// TwinCAT 3 PLC project PLC1
// ProgramVersion: 3.1.4023.0
// libraries:
//   Tc2_MC2, * (Beckhoff Automation GmbH)
//   Tc2_MC2_Drive, * (Beckhoff Automation GmbH)
//   Tc2_NcFifoAxes, * (Beckhoff Automation GmbH)
//   Tc2_Standard, * (Beckhoff Automation GmbH)
//   Tc2_System, * (Beckhoff Automation GmbH)
//   Tc2_Utilities, * (Beckhoff Automation GmbH)
//   Tc3_Module, * (Beckhoff Automation GmbH)
// project tree:
//   DUTs/ ST_streamOutputs.TcDUT
//   / PlcTask.TcTTO
//   POUs/ AxisBase.TcPOU, DigitalOut.TcPOU, FB_Fifo.TcPOU, FB_methods.TcPOU, FB_SetPositionBiasInNc_v1_10.TcPOU, FIFOaxis.TcPOU, FIFOIntegrate.TcPOU, IO.TcPOU, MAIN.TcPOU
// real-time tasks:
//   TASK PlcTask: cycle T#1ms, priority 20, ADS port 350
// motion (NC):
//   TASK NC-Task 1 SAF: cycle T#500us, priority 4, ADS port 501
//   TASK NC-Task 1 SVB: cycle T#1ms, priority 8, ADS port 511
//   AXIS motor_x1 (id 20)
//     OtherSettings: AllowMotionCmdToSlave=true, DataPersistence=true
//     encoder EncType=1
//     drive DrvType=5
//       Analog: TorqueSetpointScale=10, ScaleFactorActTorque=0.1
//       TimeComp: TaskDelayCycles=1
//     controller CtrType=1
//       CtrPara: PriorControlFactor=1
//         Observer: BandWidth=20
//   AXIS motor_x0 (id 1)
//     OtherSettings: AllowMotionCmdToSlave=true, DataPersistence=true
//     encoder EncType=1
//     drive DrvType=5
//       Analog: TorqueSetpointScale=10, ScaleFactorActTorque=0.1
//       TimeComp: TaskDelayCycles=1
//     controller CtrType=1
//       CtrPara: PriorControlFactor=1
//         Observer: BandWidth=20
//   AXIS motor_y0 (id 2)
//     OtherSettings: AllowMotionCmdToSlave=true, DataPersistence=true
//     encoder EncType=1
//     drive DrvType=5
//       Analog: TorqueSetpointScale=10, ScaleFactorActTorque=0.1
//       TimeComp: TaskDelayCycles=1
//     controller CtrType=1
//       CtrPara: PriorControlFactor=1
//         Observer: BandWidth=20
//   AXIS motor_y1 (id 3)
//     OtherSettings: AllowMotionCmdToSlave=true, DataPersistence=true
//     encoder EncType=1
//     drive DrvType=5
//       Analog: TorqueSetpointScale=10, ScaleFactorActTorque=0.1
//       TimeComp: TaskDelayCycles=1
//     controller CtrType=1
//       CtrPara: PriorControlFactor=1
//         Observer: BandWidth=20
//   AXIS motor_z1 (id 21)
//     OtherSettings: AllowMotionCmdToSlave=true, DataPersistence=true
//     encoder EncType=1
//     drive DrvType=5
//       Analog: TorqueSetpointScale=10, ScaleFactorActTorque=0.1
//       TimeComp: TaskDelayCycles=1
//     controller CtrType=1
//       CtrPara: PriorControlFactor=1
//         Observer: BandWidth=20
//   AXIS motor_z0 (id 4)
//     OtherSettings: AllowMotionCmdToSlave=true, DataPersistence=true
//     encoder EncType=1
//     drive DrvType=5
//       Analog: TorqueSetpointScale=10, ScaleFactorActTorque=0.1
//       TimeComp: TaskDelayCycles=1
//     controller CtrType=1
//       CtrPara: PriorControlFactor=1
//         Observer: BandWidth=20
//   AXIS motor_a0 (id 5)
//     OtherSettings: AllowMotionCmdToSlave=true, DataPersistence=true
//     encoder EncType=1
//     drive DrvType=5
//       Analog: TorqueSetpointScale=10, ScaleFactorActTorque=0.1
//       TimeComp: TaskDelayCycles=1
//     controller CtrType=1
//       CtrPara: PriorControlFactor=1
//         Observer: BandWidth=20
//   AXIS motor_b0 (id 6)
//     OtherSettings: AllowMotionCmdToSlave=true, DataPersistence=true
//     encoder EncType=1
//     drive DrvType=5
//       Analog: TorqueSetpointScale=10, ScaleFactorActTorque=0.1
//       TimeComp: TaskDelayCycles=1
//     controller CtrType=1
//       CtrPara: PriorControlFactor=1
//         Observer: BandWidth=20
//   AXIS motor_c0 (id 7)
//     OtherSettings: AllowMotionCmdToSlave=true, DataPersistence=true
//     encoder EncType=1
//     drive DrvType=5
//       Analog: TorqueSetpointScale=10, ScaleFactorActTorque=0.1
//       TimeComp: TaskDelayCycles=1
//     controller CtrType=1
//       CtrPara: PriorControlFactor=1
//         Observer: BandWidth=20
//   AXIS motor_d0 (id 8)
//     OtherSettings: AllowMotionCmdToSlave=true, DataPersistence=true
//     encoder EncType=1
//     drive DrvType=5
//       Analog: TorqueSetpointScale=10, ScaleFactorActTorque=0.1
//       TimeComp: TaskDelayCycles=1
//     controller CtrType=1
//       CtrPara: PriorControlFactor=1
//         Observer: BandWidth=20
//   AXIS motor_e0 (id 9)
//     OtherSettings: AllowMotionCmdToSlave=true, DataPersistence=true
//     encoder EncType=1
//     drive DrvType=5
//       Analog: TorqueSetpointScale=10, ScaleFactorActTorque=0.1
//       TimeComp: TaskDelayCycles=1
//     controller CtrType=1
//       CtrPara: PriorControlFactor=1
//         Observer: BandWidth=20
//   AXIS motor_x_master (id 10)
//     OtherSettings: AllowMotionCmdToSlave=true
//     encoder EncType=1
//     drive DrvType=5
//       Analog: TorqueSetpointScale=10, ScaleFactorActTorque=0.1
//       TimeComp: TaskDelayCycles=1
//     controller CtrType=1
//       CtrPara: PriorControlFactor=1
//         Observer: BandWidth=20
//   AXIS motor_y_master (id 11)
//     OtherSettings: AllowMotionCmdToSlave=true
//     encoder EncType=1
//     drive DrvType=5
//       Analog: TorqueSetpointScale=10, ScaleFactorActTorque=0.1
//       TimeComp: TaskDelayCycles=1
//     controller CtrType=1
//       CtrPara: PriorControlFactor=1
//         Observer: BandWidth=20
//   AXIS motor_z_master (id 12)
//     OtherSettings: AllowMotionCmdToSlave=true
//     encoder EncType=1
//     drive DrvType=5
//       Analog: TorqueSetpointScale=10, ScaleFactorActTorque=0.1
//       TimeComp: TaskDelayCycles=1
//     controller CtrType=1
//       CtrPara: PriorControlFactor=1
//         Observer: BandWidth=20
//   AXIS motor_a_master (id 13)
//     OtherSettings: AllowMotionCmdToSlave=true
//     encoder EncType=1
//     drive DrvType=5
//       Analog: TorqueSetpointScale=10, ScaleFactorActTorque=0.1
//       TimeComp: TaskDelayCycles=1
//     controller CtrType=1
//       CtrPara: PriorControlFactor=1
//         Observer: BandWidth=20
//   AXIS motor_b_master (id 14)
//     OtherSettings: AllowMotionCmdToSlave=true
//     encoder EncType=1
//     drive DrvType=5
//       Analog: TorqueSetpointScale=10, ScaleFactorActTorque=0.1
//       TimeComp: TaskDelayCycles=1
//     controller CtrType=1
//       CtrPara: PriorControlFactor=1
//         Observer: BandWidth=20
//   AXIS motor_c_master (id 15)
//     OtherSettings: AllowMotionCmdToSlave=true
//     encoder EncType=1
//     drive DrvType=5
//       Analog: TorqueSetpointScale=10, ScaleFactorActTorque=0.1
//       TimeComp: TaskDelayCycles=1
//     controller CtrType=1
//       CtrPara: PriorControlFactor=1
//         Observer: BandWidth=20
//   AXIS motor_d_master (id 16)
//     OtherSettings: AllowMotionCmdToSlave=true
//     encoder EncType=1
//     drive DrvType=5
//       Analog: TorqueSetpointScale=10, ScaleFactorActTorque=0.1
//       TimeComp: TaskDelayCycles=1
//     controller CtrType=1
//       CtrPara: PriorControlFactor=1
//         Observer: BandWidth=20
//   AXIS motor_e_master (id 17)
//     OtherSettings: AllowMotionCmdToSlave=true
//     encoder EncType=1
//     drive DrvType=5
//       Analog: TorqueSetpointScale=10, ScaleFactorActTorque=0.1
//       TimeComp: TaskDelayCycles=1
//     controller CtrType=1
//       CtrPara: PriorControlFactor=1
//         Observer: BandWidth=20
//   AXIS motor_z1_multimaster (id 22)
//     OtherSettings: AllowMotionCmdToSlave=true
//     encoder EncType=1
//     drive DrvType=5
//       Analog: TorqueSetpointScale=10, ScaleFactorActTorque=0.1
//       TimeComp: TaskDelayCycles=1
//     controller CtrType=1
//       CtrPara: PriorControlFactor=1
//         Observer: BandWidth=20
//   AXIS motor_z0_multimaster (id 18)
//     OtherSettings: AllowMotionCmdToSlave=true
//     encoder EncType=1
//     drive DrvType=5
//       Analog: TorqueSetpointScale=10, ScaleFactorActTorque=0.1
//       TimeComp: TaskDelayCycles=1
//     controller CtrType=1
//       CtrPara: PriorControlFactor=1
//         Observer: BandWidth=20
//   AXIS motor_z1_masterOffset (id 23)
//     OtherSettings: AllowMotionCmdToSlave=true
//     encoder EncType=1
//     drive DrvType=5
//       Analog: TorqueSetpointScale=10, ScaleFactorActTorque=0.1
//       TimeComp: TaskDelayCycles=1
//     controller CtrType=1
//       CtrPara: PriorControlFactor=1
//         Observer: BandWidth=20
//   AXIS motor_z0_masterOffset (id 19)
//     OtherSettings: AllowMotionCmdToSlave=true
//     encoder EncType=1
//     drive DrvType=5
//       Analog: TorqueSetpointScale=10, ScaleFactorActTorque=0.1
//       TimeComp: TaskDelayCycles=1
//     controller CtrType=1
//       CtrPara: PriorControlFactor=1
//         Observer: BandWidth=20
// variable links:
//   PLC1/PLC1 Instance <-> NC-Task 1 SAF/Axes/motor_a0
//     PlcTask Inputs/MAIN.motor_a0.axis.NcToPlc <-> Outputs/ToPlc
//     PlcTask Outputs/MAIN.motor_a0.axis.PlcToNc <-> Inputs/FromPlc
//   PLC1/PLC1 Instance <-> NC-Task 1 SAF/Axes/motor_a_master
//     PlcTask Inputs/MAIN.motor_a_master.axis.NcToPlc <-> Outputs/ToPlc
//     PlcTask Outputs/MAIN.motor_a_master.axis.PlcToNc <-> Inputs/FromPlc
//   PLC1/PLC1 Instance <-> NC-Task 1 SAF/Axes/motor_b0
//     PlcTask Inputs/MAIN.motor_b0.axis.NcToPlc <-> Outputs/ToPlc
//     PlcTask Outputs/MAIN.motor_b0.axis.PlcToNc <-> Inputs/FromPlc
//   PLC1/PLC1 Instance <-> NC-Task 1 SAF/Axes/motor_b_master
//     PlcTask Inputs/MAIN.motor_b_master.axis.NcToPlc <-> Outputs/ToPlc
//     PlcTask Outputs/MAIN.motor_b_master.axis.PlcToNc <-> Inputs/FromPlc
//   PLC1/PLC1 Instance <-> NC-Task 1 SAF/Axes/motor_c0
//     PlcTask Inputs/MAIN.motor_c0.axis.NcToPlc <-> Outputs/ToPlc
//     PlcTask Outputs/MAIN.motor_c0.axis.PlcToNc <-> Inputs/FromPlc
//   PLC1/PLC1 Instance <-> NC-Task 1 SAF/Axes/motor_c_master
//     PlcTask Inputs/MAIN.motor_c_master.axis.NcToPlc <-> Outputs/ToPlc
//     PlcTask Outputs/MAIN.motor_c_master.axis.PlcToNc <-> Inputs/FromPlc
//   PLC1/PLC1 Instance <-> NC-Task 1 SAF/Axes/motor_d0
//     PlcTask Inputs/MAIN.motor_d0.axis.NcToPlc <-> Outputs/ToPlc
//     PlcTask Outputs/MAIN.motor_d0.axis.PlcToNc <-> Inputs/FromPlc
//   PLC1/PLC1 Instance <-> NC-Task 1 SAF/Axes/motor_d_master
//     PlcTask Inputs/MAIN.motor_d_master.axis.NcToPlc <-> Outputs/ToPlc
//     PlcTask Outputs/MAIN.motor_d_master.axis.PlcToNc <-> Inputs/FromPlc
//   PLC1/PLC1 Instance <-> NC-Task 1 SAF/Axes/motor_e0
//     PlcTask Inputs/MAIN.motor_e0.axis.NcToPlc <-> Outputs/ToPlc
//     PlcTask Outputs/MAIN.motor_e0.axis.PlcToNc <-> Inputs/FromPlc
//   PLC1/PLC1 Instance <-> NC-Task 1 SAF/Axes/motor_e_master
//     PlcTask Inputs/MAIN.motor_e_master.axis.NcToPlc <-> Outputs/ToPlc
//     PlcTask Outputs/MAIN.motor_e_master.axis.PlcToNc <-> Inputs/FromPlc
//   PLC1/PLC1 Instance <-> NC-Task 1 SAF/Axes/motor_x0
//     PlcTask Inputs/MAIN.motor_x0.axis.NcToPlc <-> Outputs/ToPlc
//     PlcTask Outputs/MAIN.motor_x0.axis.PlcToNc <-> Inputs/FromPlc
//   PLC1/PLC1 Instance <-> NC-Task 1 SAF/Axes/motor_x1
//     PlcTask Inputs/MAIN.motor_x1.axis.NcToPlc <-> Outputs/ToPlc
//     PlcTask Outputs/MAIN.motor_x1.axis.PlcToNc <-> Inputs/FromPlc
//   PLC1/PLC1 Instance <-> NC-Task 1 SAF/Axes/motor_x_master
//     PlcTask Inputs/MAIN.motor_x_master.axis.NcToPlc <-> Outputs/ToPlc
//     PlcTask Outputs/MAIN.motor_x_master.axis.PlcToNc <-> Inputs/FromPlc
//   PLC1/PLC1 Instance <-> NC-Task 1 SAF/Axes/motor_y0
//     PlcTask Inputs/MAIN.motor_y0.axis.NcToPlc <-> Outputs/ToPlc
//     PlcTask Outputs/MAIN.motor_y0.axis.PlcToNc <-> Inputs/FromPlc
//   PLC1/PLC1 Instance <-> NC-Task 1 SAF/Axes/motor_y1
//     PlcTask Inputs/MAIN.motor_y1.axis.NcToPlc <-> Outputs/ToPlc
//     PlcTask Outputs/MAIN.motor_y1.axis.PlcToNc <-> Inputs/FromPlc
//   PLC1/PLC1 Instance <-> NC-Task 1 SAF/Axes/motor_y_master
//     PlcTask Inputs/MAIN.motor_y_master.axis.NcToPlc <-> Outputs/ToPlc
//     PlcTask Outputs/MAIN.motor_y_master.axis.PlcToNc <-> Inputs/FromPlc
//   PLC1/PLC1 Instance <-> NC-Task 1 SAF/Axes/motor_z0
//     PlcTask Inputs/MAIN.motor_z0.axis.NcToPlc <-> Outputs/ToPlc
//     PlcTask Outputs/MAIN.motor_z0.axis.PlcToNc <-> Inputs/FromPlc
//   PLC1/PLC1 Instance <-> NC-Task 1 SAF/Axes/motor_z0_masterOffset
//     PlcTask Inputs/MAIN.motor_z0_master_offset.axis.NcToPlc <-> Outputs/ToPlc
//     PlcTask Outputs/MAIN.motor_z0_master_offset.axis.PlcToNc <-> Inputs/FromPlc
//   PLC1/PLC1 Instance <-> NC-Task 1 SAF/Axes/motor_z0_multimaster
//     PlcTask Inputs/MAIN.motor_z0_multimaster.axis.NcToPlc <-> Outputs/ToPlc
//     PlcTask Outputs/MAIN.motor_z0_multimaster.axis.PlcToNc <-> Inputs/FromPlc
//   PLC1/PLC1 Instance <-> NC-Task 1 SAF/Axes/motor_z1
//     PlcTask Inputs/MAIN.motor_z1.axis.NcToPlc <-> Outputs/ToPlc
//     PlcTask Outputs/MAIN.motor_z1.axis.PlcToNc <-> Inputs/FromPlc
//   PLC1/PLC1 Instance <-> NC-Task 1 SAF/Axes/motor_z1_masterOffset
//     PlcTask Inputs/MAIN.motor_z1_master_offset.axis.NcToPlc <-> Outputs/ToPlc
//     PlcTask Outputs/MAIN.motor_z1_master_offset.axis.PlcToNc <-> Inputs/FromPlc
//   PLC1/PLC1 Instance <-> NC-Task 1 SAF/Axes/motor_z1_multimaster
//     PlcTask Inputs/MAIN.motor_z1_multimaster.axis.NcToPlc <-> Outputs/ToPlc
//     PlcTask Outputs/MAIN.motor_z1_multimaster.axis.PlcToNc <-> Inputs/FromPlc
//   PLC1/PLC1 Instance <-> NC-Task 1 SAF/Axes/motor_z_master
//     PlcTask Inputs/MAIN.motor_z_master.axis.NcToPlc <-> Outputs/ToPlc
//     PlcTask Outputs/MAIN.motor_z_master.axis.PlcToNc <-> Inputs/FromPlc

CONFIGURATION PLC1
    RESOURCE PLC ON TwinCAT3
        TASK PlcTask(INTERVAL := T#1ms, PRIORITY := 20);
        PROGRAM MAIN WITH PlcTask : MAIN;
    END_RESOURCE
END_CONFIGURATION

// ---- DUTs/ST_streamOutputs.TcDUT
TYPE ST_streamOutputs :
STRUCT
	cycleNo : UDINT;
	on : BOOL;

END_STRUCT
END_TYPE

// ---- POUs/MAIN.TcPOU
PROGRAM MAIN
VAR
	motor_x0 : AxisBase;
	motor_x1 : AxisBase;	
	motor_y0 : AxisBase;
	motor_y1 : AxisBase;
	motor_z0 : AxisBase;
	motor_z1 : AxisBase;	
	motor_a0 : AxisBase;
	motor_b0 : AxisBase;
	motor_c0 : AxisBase;
	motor_d0 : AxisBase;
	motor_e0 : AxisBase;
	
	motor_x_master : AxisBase;
	motor_y_master : AxisBase;
	motor_z_master : AxisBase;
	motor_a_master : AxisBase;
	motor_b_master : AxisBase;
	motor_c_master : AxisBase;
	motor_d_master : AxisBase;
	motor_e_master : AxisBase;
	
	motor_z0_master_offset : AxisBase;
	motor_z0_multimaster : AxisBase;
	motor_z1_master_offset : AxisBase;
	motor_z1_multimaster : AxisBase;
	emptyAxis1 : AXIS_REF;
	emptyAxis2 : AXIS_REF;

	gearOutAll: BOOL;
	n: INT;
	
	fbMultiMaster_z0 : MC_GearInMultiMaster;
	fbPower_multimaster : MC_Power;
	fbPower_z0_offset : MC_Power;
	bStartMultiMaster_z0: BOOL;
	fbGearOutMulti_z0 : MC_GearOut;
	
	fbMultiMaster_z1 : MC_GearInMultiMaster;
	fbPower_multimaster_z1 : MC_Power;
	fbPower_z1_offset : MC_Power;
	bStartMultiMaster_z1: BOOL;
	fbGearOutMulti_z1 : MC_GearOut;
	
	
	geartest : MC_GearIn;
	
	fbSystemTime : GETSYSTEMTIME;
	fileTime        : T_FILETIME;

	sTimeString: STRING(24);
	ppp: INT;
END_VAR


ppp := ppp + 1;


fbSystemTime(timeLoDW => fileTime.dwLowDateTime, timeHiDW => fileTime.dwHighDateTime );
sTimeString := SYSTEMTIME_TO_STRING(FILETIME_TO_SYSTEMTIME(fileTime));

FIFOaxis();

IO();


motor_x0(bPower:= , bMoveAbs:= , bMoveVel:= , bPowerStatus=> );
motor_x1(bPower:= , bMoveAbs:= , bMoveVel:= , bPowerStatus=> );
motor_y0(bPower:= , bMoveAbs:= , bMoveVel:= , bPowerStatus=> );
motor_y1(bPower:= , bMoveAbs:= , bMoveVel:= , bPowerStatus=> );
motor_z0(bPower:= , bMoveAbs:= , bMoveVel:= , bPowerStatus=> );
motor_z1(bPower:= , bMoveAbs:= , bMoveVel:= , bPowerStatus=> );
motor_a0(bPower:= , bMoveAbs:= , bMoveVel:= , bPowerStatus=> );
motor_b0(bPower:= , bMoveAbs:= , bMoveVel:= , bPowerStatus=> );
motor_c0(bPower:= , bMoveAbs:= , bMoveVel:= , bPowerStatus=> );
motor_d0(bPower:= , bMoveAbs:= , bMoveVel:= , bPowerStatus=> );
motor_e0(bPower:= , bMoveAbs:= , bMoveVel:= , bPowerStatus=> );

motor_x_master(bPower:= , bMoveAbs:= , bMoveVel:= , bPowerStatus=> );
motor_y_master(bPower:= , bMoveAbs:= , bMoveVel:= , bPowerStatus=> );
motor_z_master(bPower:= , bMoveAbs:= , bMoveVel:= , bPowerStatus=> );
motor_a_master(bPower:= , bMoveAbs:= , bMoveVel:= , bPowerStatus=> );
motor_b_master(bPower:= , bMoveAbs:= , bMoveVel:= , bPowerStatus=> );
motor_c_master(bPower:= , bMoveAbs:= , bMoveVel:= , bPowerStatus=> );
motor_d_master(bPower:= , bMoveAbs:= , bMoveVel:= , bPowerStatus=> );
motor_e_master(bPower:= , bMoveAbs:= , bMoveVel:= , bPowerStatus=> );

motor_z0_multimaster(bPower:= , bMoveAbs:= , bMoveVel:= , bPowerStatus=> );
motor_z0_master_offset(bPower:= , bMoveAbs:= , bMoveVel:= , bPowerStatus=> );
motor_z1_multimaster(bPower:= , bMoveAbs:= , bMoveVel:= , bPowerStatus=> );
motor_z1_master_offset(bPower:= , bMoveAbs:= , bMoveVel:= , bPowerStatus=> );




IF fbGearOutMulti_z0.Execute AND NOT fbGearOutMulti_z0.Busy THEN
	fbGearOutMulti_z0.Execute := FALSE;
END_IF
IF fbGearOutMulti_z1.Execute AND NOT fbGearOutMulti_z1.Busy THEN
	fbGearOutMulti_z1.Execute := FALSE;
END_IF

IF gearOutAll THEN
	bStartMultiMaster_z0 := FALSE;
	bStartMultiMaster_z1 := FALSE;	
	motor_x0.M_GearOut('motor_x0');
	motor_x1.M_GearOut('motor_x0');
	motor_y0.M_GearOut('motor_y0');
	motor_y1.M_GearOut('motor_y1');
	motor_z0.M_GearOut('motor_z0');
	motor_z1.M_GearOut('motor_z0');	
	motor_a0.M_GearOut('motor_a0');
	motor_b0.M_GearOut('motor_b0');
	motor_c0.M_GearOut('motor_c0');
	motor_d0.M_GearOut('motor_d0');
	motor_e0.M_GearOut('motor_e0');
	fbGearOutMulti_z0.Execute := TRUE;	
	fbGearOutMulti_z1.Execute := TRUE;	
	gearOutAll := FALSE;
END_IF




	
//multimaster, för z0-axel


fbMultiMaster_z0(
	Master1:= motor_z0_master_offset.axis, 
	Master2:= motor_z_master.axis, 
	Master3:= emptyAxis1, 
	Master4:= emptyAxis2, 
	Slave:= motor_z0_multimaster.axis, 
	Enable:= bStartMultiMaster_z0, 
	GearRatio1:= 1, 
	GearRatio2:= 1, 
	GearRatio3:= 0, 
	GearRatio4:= 0, 
	Acceleration:= , 
	Deceleration:= , 
	Jerk:= , 
	BufferMode:= , 
	Options:= , 
	InGear=> , 
	Busy=> , 
	Active=> , 
	CommandAborted=> , 
	Error=> , 
	ErrorID=> );

fbPower_multimaster(
	Axis:= motor_z0_multimaster.axis, 
	Enable:= TRUE, 
	Enable_Positive:= TRUE, 
	Enable_Negative:= TRUE, 
	Override:= , 
	BufferMode:= , 
	Options:= , 
	Status=> , 
	Busy=> , 
	Active=> , 
	Error=> , 
	ErrorID=> );

fbPower_z0_offset(
	Axis:= motor_z0_master_offset.axis, 
	Enable:= TRUE, 
	Enable_Positive:= TRUE, 
	Enable_Negative:= TRUE, 
	Override:= , 
	BufferMode:= , 
	Options:= , 
	Status=> , 
	Busy=> , 
	Active=> , 
	Error=> , 
	ErrorID=> );

fbGearOutMulti_z0(
	Slave:= motor_z0_multimaster.axis, 
	Execute:= , 
	Options:= , 
	Done=> , 
	Busy=> , 
	Error=> , 
	ErrorID=> );
	
	
//multimaster, för z1-axel


fbMultiMaster_z1(
	Master1:= motor_z1_master_offset.axis, 
	Master2:= motor_z_master.axis, 
	Master3:= emptyAxis1, 
	Master4:= emptyAxis2, 
	Slave:= motor_z1_multimaster.axis, 
	Enable:= bStartMultiMaster_z1, 
	GearRatio1:= 1, 
	GearRatio2:= 1, 
	GearRatio3:= 0, 
	GearRatio4:= 0, 
	Acceleration:= , 
	Deceleration:= , 
	Jerk:= , 
	BufferMode:= , 
	Options:= , 
	InGear=> , 
	Busy=> , 
	Active=> , 
	CommandAborted=> , 
	Error=> , 
	ErrorID=> );

fbPower_multimaster_z1(
	Axis:= motor_z1_multimaster.axis, 
	Enable:= TRUE, 
	Enable_Positive:= TRUE, 
	Enable_Negative:= TRUE, 
	Override:= , 
	BufferMode:= , 
	Options:= , 
	Status=> , 
	Busy=> , 
	Active=> , 
	Error=> , 
	ErrorID=> );

fbPower_z1_offset(
	Axis:= motor_z1_master_offset.axis, 
	Enable:= TRUE, 
	Enable_Positive:= TRUE, 
	Enable_Negative:= TRUE, 
	Override:= , 
	BufferMode:= , 
	Options:= , 
	Status=> , 
	Busy=> , 
	Active=> , 
	Error=> , 
	ErrorID=> );

fbGearOutMulti_z1(
	Slave:= motor_z1_multimaster.axis, 
	Execute:= , 
	Options:= , 
	Done=> , 
	Busy=> , 
	Error=> , 
	ErrorID=> );

METHOD M_GearOutAll : BOOL
VAR_INPUT
END_VAR
gearOutAll := TRUE;
END_METHOD

END_PROGRAM

// ---- POUs/AxisBase.TcPOU
FUNCTION_BLOCK AxisBase
VAR_INPUT
	bPower : BOOL;
	bMoveAbs : BOOL;
	bMoveVel : BOOL;

END_VAR
VAR_OUTPUT
	bPowerStatus : BOOL;
END_VAR
VAR
	isVirtual : BOOL;
	axis : AXIS_REF;
	fPosition : LREAL;		//from cnc
	fVelocity : LREAL;		//from cnc
	fAcc : LREAL;			//from cnc
	fDeacc : LREAL; 			//from cnc
	fbAxisPower : MC_Power;
	fbMoveAbsolute : MC_MoveAbsolute;
	fbHalt : MC_Halt;
	fbMoveVelocity : MC_MoveVelocity;
	axisState: INT;
	pp: INT;
	p: INT;
	fbGearIn : ARRAY[1..9] OF MC_GearIn;
	fbGearOut : MC_GearOut;
	a: INT;
	fbHome : MC_Home;
	fbHomeMemory: FB_CoEAX8000SetPositionOffset;  
	fbBias : FB_SetPositionBiasInNc_v1_10;  
	HomePos: LREAL;
	HomeSeq: INT;
	StartHome: BOOL;
	AxisHomed : BOOL;
	
	//torque
	MaxTorque : LREAL;
	MinTorque : LREAL;
	fbSoEread : FB_SoERead;
	
	axisIsGeared : BOOL;
	goBacktoFifo: BOOL;
	
	//reset
	fbReset : MC_Reset;
	b: INT;
	c: INT;
	fBias: LREAL;
	aa: INT;
	HomeSeqMemory: INT;
	StartHomeMemory: BOOL;
	bAxisDriveError: BOOL;
	bAxisError: BOOL;
END_VAR


axis.ReadStatus();
bAxisError:=axis.Status.Error;
bAxisDriveError:=axis.Status.DriveDeviceError;


CASE axisState OF

0:
	IF bMoveAbs THEN
		axisState := 100;
		b := b +1;
	END_IF
	IF bMoveVel THEN
		c := c +1;
		axisState := 200;
	END_IF

10:
	IF FIFOaxis.FifoActive THEN 
		goBacktoFifo := TRUE;
		MAIN.M_gearOutAll();
	END_IF	
	axisState := 20;

20:
	IF FIFOaxis.FifoActive THEN 
		FIFOaxis.M_deIntegrate();
	END_IF
	axisState := 30;
	

	
100:
	fbHalt.Execute := TRUE;
	IF (fbHalt.Busy AND NOT fbMoveAbsolute.Busy) OR fbHalt.Done THEN
		fbHalt.Execute := FALSE;
		axisState := 120;
	END_IF		

	
120:
	bMoveAbs := FALSE;	
	IF fVelocity <> 0 THEN
	fbmoveAbsolute.Execute := TRUE;
		axisState := 130;
	ELSE
		axisState := 0;
	END_IF
	
130:
	IF fbMoveAbsolute.Busy THEN
		fbMoveAbsolute.Execute := FALSE;
		axisState := 140;
	END_IF
	pp := pp +1;

140: 
	axisState := 0;	



200:
	fbHalt.Execute := TRUE;
	axisState := 210;

210:
	fbHalt.Execute := FALSE;
	axisState := 220;
	
220:
	bMoveVel := FALSE;
	IF fVelocity <> 0 THEN
		fbMoveVelocity.Execute := TRUE;	
		axisState := 230;
	ELSE
		axisState := 0;
	END_IF
	
230: 
	fbMoveVelocity.Execute := FALSE;
	axisState := 0;	


END_CASE





fbMoveAbsolute(
	Axis:= axis, 
	Execute:= , 
	Position:= fPosition, 
	Velocity:= fVelocity, 
	Acceleration:= fAcc, 
	Deceleration:= fDeacc, 
	Jerk:= 1000, 
	BufferMode:= ,//MC_BufferMode.MC_Aborting, 
	Options:= , 
	Done=> , 
	Busy=> , 
	Active=> , 
	CommandAborted=> , 
	Error=> , 
	ErrorID=> );
	
	
fbMoveVelocity(
	Axis:= axis, 
	Execute:= , 
	Velocity:= fVelocity, 
	Acceleration:= fAcc, 
	Deceleration:= fDeacc, 
	Jerk:= 5000, 
	Direction:= , 
	BufferMode:= , 
	Options:= , 
	InVelocity=> , 
	Busy=> , 
	Active=> , 
	CommandAborted=> , 
	Error=> , 
	ErrorID=> );

	
fbHalt(
	Axis:= axis, 
	Execute:= , 
	Deceleration:= 1000, 
	Jerk:= 5000, 
	BufferMode:= , 
	Options:= , 
	Done=> , 
	Busy=> , 
	Active=> , 
	CommandAborted=> , 
	Error=> , 
	ErrorID=> );

	
fbAxisPower(
	Axis:= axis, 
	Enable:= bPower, 
	Enable_Positive:= TRUE, 
	Enable_Negative:= TRUE, 
	Override:= 100, 
	BufferMode:= ,
	Options:= , 
	Status=> bPowerStatus, 
	Busy=> , 
	Active=> , 
	Error=> , 
	ErrorID=> );
	

	//GEAR

FOR a:=1 TO 9 DO
	IF fbGearIn[a].Execute AND fbGearIn[a].Busy THEN 
		fbGearIn[a].Execute := FALSE; 
	END_IF
END_FOR


IF fbGearOut.Execute AND fbGearOut.Busy THEN
	fbhalt.Execute := FALSE;
	fbGearOut.Execute := FALSE;
END_IF



	
fbGearOut(
	Slave:= axis, 
	Execute:= , 
	Options:= , 
	Done=> , 
	Busy=> , 
	Error=> , 
	ErrorID=> );

fbGearIn[1](Master:= main.motor_x_master.axis, Slave:= axis, RatioDenominator := 1, RatioNumerator := 1);
fbGearIn[2](Master:= main.motor_y_master.axis, Slave:= axis, RatioDenominator := 1, RatioNumerator := 1);
fbGearIn[3](Master:= main.motor_z0_multimaster.axis, Slave:= axis, RatioDenominator := 1, RatioNumerator := 1);
fbGearIn[4](Master:= main.motor_a_master.axis, Slave:= axis, RatioDenominator := 1, RatioNumerator := 1);
fbGearIn[5](Master:= main.motor_b_master.axis, Slave:= axis, RatioDenominator := 1, RatioNumerator := 1);
fbGearIn[6](Master:= main.motor_c_master.axis, Slave:= axis, RatioDenominator := 1, RatioNumerator := 1);
fbGearIn[7](Master:= main.motor_d_master.axis, Slave:= axis, RatioDenominator := 1, RatioNumerator := 1);
fbGearIn[8](Master:= main.motor_e_master.axis, Slave:= axis, RatioDenominator := 1, RatioNumerator := 1);
fbGearIn[9](Master:= main.motor_z1_multimaster.axis, Slave:= axis, RatioDenominator := 1, RatioNumerator := 1);	
	
//HOMING

CASE HomeSeq OF
	
	0: 
		IF 	StartHome THEN
			HomeSeq := 10;
		END_IF

		
	10:
		StartHome := FALSE;
		fbHome.Position := HomePos;
		HomeSeq := 20;
				aa := aa +1;
	20:
		fbHome.Execute := TRUE;
		//fbBias.bExecute :=TRUE;
		HomeSeq := 30;
		
	30:
		IF fbHome.Execute AND NOT fbHome.Busy THEN
			fbHome.Execute := FALSE;
			//fbBias.bExecute :=FALSE;
			HomeSeq :=0;
			AxisHomed := TRUE;
		END_IF

END_CASE


CASE HomeSeqMemory OF
	
	0: 
		IF 	StartHomeMemory THEN
			HomeSeqMemory := 10;
		END_IF

		
	10:
		StartHomeMemory := FALSE;
		fbHomeMemory.Position := HomePos;
		fbHomeMemory.Memory := 1;
		fbHomeMemory.Feedback := 0;
		HomeSeqMemory := 20;
	
	20:
		fbHomeMemory.Execute := TRUE;
		//fbBias.bExecute :=TRUE;
		HomeSeqMemory := 30;
		
	30:
		IF fbHomeMemory.Execute AND NOT fbHomeMemory.Busy THEN
			fbHomeMemory.Execute := FALSE;
			//fbBias.bExecute :=FALSE;
			HomeSeqMemory :=0;
			//AxisHomed := TRUE;
		END_IF

END_CASE


fbHome(
	Axis:= axis, 
	Execute:= , 
	Position:= , 
	HomingMode:= MC_HomingMode.MC_Direct, 
	BufferMode:= , 
	Options:= , 
	bCalibrationCam:= , 
	Done=> , 
	Busy=> , 
	Active=> , 
	CommandAborted=> , 
	Error=> , 
	ErrorID=> );
	

fBias := (HomePos - axis.NcToPlc.ActPos);
fbBias(
	bInit:= , 
	bExecute:= , 
	fOffset:= , 
	bBusy=> , 
	bDone=> , 
	bError=> , 
	nErrorId=> , 
	fPositionBias:= fBias, 
	Axis:= axis);
	

	// TORQUE
	//ska läsas skriva till driven. Olika för olika typer av drives. Ex Sercos:
	
	fbSoEread(
	Axis:= axis, 
	NetId:= '', 
	Idn:= S_0_IDNs + 82, 
	Element:= 16#40, 
	pDstBuf:= ADR(MaxTorque), 
	BufLen:= SIZEOF(MaxTorque), 
	Execute:= , 
	Timeout:= , 
	Busy=> , 
	Error=> , 
	AdsErrId=> , 
	SercosErrId=> , 
	Attribute=> );
	

IF fbReset.Execute AND fbReset.Busy THEN
	fbReset.Execute := FALSE;
END_IF

	
fbReset(
	Axis:= axis, 
	Execute:= , 
	Done=> , 
	Busy=> , 
	Error=> , 
	ErrorID=> );

{attribute 'TcRpcEnable'}
METHOD M_GearIn : BOOL
VAR_INPUT
	Slavename : STRING;
	Master : int;
END_VAR

axisIsGeared := TRUE;


IF (master = 1) THEN
	fbGearIn[1].Execute := TRUE;
ELSIF (master = 2) THEN
	fbGearIn[2].Execute := TRUE;
ELSIF (master = 3) THEN
	fbGearIn[3].Execute := TRUE;
ELSIF (master = 4) THEN
	fbGearIn[4].Execute := TRUE;
ELSIF (master = 5) THEN
	fbGearIn[5].Execute := TRUE;
ELSIF (master = 6) THEN
	fbGearIn[6].Execute := TRUE;
ELSIF (master = 7) THEN
	fbGearIn[7].Execute := TRUE;
ELSIF (master = 8) THEN
	fbGearIn[8].Execute := TRUE;
ELSIF (master = 9) THEN
	fbGearIn[9].Execute := TRUE;
ELSE
	//
END_IF
END_METHOD

{attribute 'TcRpcEnable'}
METHOD M_GearOut : BOOL
VAR_INPUT
	slavename : STRING;
END_VAR


axisIsGeared := FALSE;
fbhalt.Execute := TRUE;

fbGearOut.Execute := TRUE;
END_METHOD

END_FUNCTION_BLOCK

// ---- POUs/FB_SetPositionBiasInNc_v1_10.TcPOU
FUNCTION_BLOCK FB_SetPositionBiasInNc_v1_10
VAR_INPUT
	bInit: BOOL;
	bExecute: BOOL;
	fOffset: LREAL;
END_VAR
VAR_OUTPUT
	bBusy: BOOL;
	bDone: BOOL;
	bError: BOOL;
	nErrorId: UDINT;
END_VAR
VAR_IN_OUT
	fPositionBias: LREAL;
	Axis: TC2_MC2.AXIS_REF;
END_VAR
VAR
	nState: UINT;
	fbADSREAD: ADSREAD;
	fbADSWRITE: ADSWRITE;
END_VAR



(*Sequence to set Position Bias in Nc*)
CASE nState OF
0: (*Start sequence. Wait until bExecute is TRUE*)
	IF bInit THEN
	bBusy:=TRUE;
	bError:=FALSE;
	nErrorId:=0;
	nState:=30;
	ELSIF bExecute THEN
	bBusy:=TRUE;
	bError:=FALSE;
	nErrorId:=0;
	nState:=10;
	END_IF



10: (*Read actual Position Bias in Nc*)
fbADSREAD(
PORT:=500,
IDXGRP:=16#5000+Axis.NcToPlc.AxisId,
IDXOFFS:=16#7,
LEN:=SIZEOF(fPositionBias),
DESTADDR:=ADR(fPositionBias),
READ:=TRUE);



(*Wait until it's done or if an error occurs*)
IF NOT fbADSREAD.ERR THEN
IF NOT fbADSREAD.BUSY THEN
fbADSREAD(READ:=FALSE);
nState:=20;
END_IF
ELSE
nErrorId:=fbADSREAD.ERRID;
nState:=999;
END_IF



20:(*Calculate new Position Bias*)
fPositionBias:=fPositionBias+((Axis.NcToPlc.ActPos-REAL_TO_LREAL(fOffset)) *-1);
nState:=30;



30: (*Write Position Bias in Nc*)
fbADSWRITE(
PORT:=500,
IDXGRP:=16#5000+Axis.NcToPlc.AxisId,
IDXOFFS:=16#7,
LEN:=SIZEOF(fPositionBias),
SRCADDR:=ADR(fPositionBias),
WRITE:=TRUE);



(*Wait until it's done or if an error occurs*)
IF NOT fbADSWRITE.ERR THEN
IF NOT fbADSWRITE.BUSY THEN
fbADSWRITE(WRITE:=FALSE);
nState:=40;
END_IF
ELSE
nErrorId:=fbADSWRITE.ERRID;
nState:=999;
END_IF



40: (*Sequense is done. Waits until bExecute is FALSE*)
bBusy:=FALSE;
bDone:=TRUE;
IF NOT (bInit OR bExecute) THEN
bDone:=FALSE;
nState:=0;
END_IF



999: (*Error in sequence*)
bError:=TRUE;
bBusy:=FALSE;
bDone:=FALSE;
fbADSREAD(READ:=FALSE);
fbADSWRITE(WRITE:=FALSE);
IF NOT (bInit OR bExecute) THEN
nState:=0;
END_IF



END_CASE

END_FUNCTION_BLOCK

// ---- POUs/FIFOaxis.TcPOU
PROGRAM FIFOaxis
VAR

	FifoOverride : FiFoSetChannelOverride;
	FifoDeIntegrate : FiFoGroupDisintegrate;
	FiFoReadDim1: FiFoGetDimension;
	FifoReadDimOK: BOOL;
	FifoNoOfAxis: UDINT;
	FifoNoOfEntries: UDINT;
	FIFOChInegrate : ARRAY[1..8] of FIFOIntegrate;
	FreeRows: DINT;
	NrOccupiedLines: DINT;
	n: UINT;
	StartIntegration: BOOL;

	FifoTableFromCNC	:	ARRAY[0..49,0..7] OF LREAL;
	FifoTableFromCNCLine:	ARRAY[0..400] OF LREAL;		//pos0 = number of rows
	FifoTableFromCNCTemp:	ARRAY[0..49,0..7] OF LREAL;
	FifoTable2	:	ARRAY[0..49,0..7] OF LREAL;

	FifoState: INT;
	StartFifo: BOOL;
	nOverride: UDINT;
	FrameNumber : UDINT;
	
	FifoWrite : FiFoWrite;
	FifoStart : FiFoStart;
	FifoStop : FifoStop;
	FifoTableCanTakeData : BOOL;
	FifoHasWritten : BOOL;
	
	m: INT;
	RowsFromCNC: UDINT;
	FiFoRunState: INT;
	p: INT;
	StartInt: INT;
	FifoActive: BOOL;
	fbMethods : FB_methods;
END_VAR


FifoStop(
	iChannelId:= 2, 
	bExecute:= , 
	tTimeout:= , 
	bBusy=> , 
	bErr=> , 
	iErrId=> );


CASE FifoState OF 
	
0:
	IF StartFifo THEN
		FrameNumber := 0;
		FifoState := 10;
	END_IF

10:
	StartIntegration := TRUE;
	StartFifo := FALSE;
	FifoOverride.bExecute := TRUE;
	FifoState := 20;

20: 
	StartIntegration := FALSE;
	FifoOverride.bExecute := FALSE;
	FiFoReadDim1.bExecute := TRUE;
	FifoState := 30;
	
30:
	FiFoReadDim1.bExecute := FALSE;
	FifoState := 40;
	
40:
	StartIntegration := TRUE;
	FifoState := 50;
	
50:
		FifoTableCanTakeData := TRUE;

		FIfostate := 100;

	
100:
	
	IF FifoHasWritten THEN
		FOR p := 0 TO LREAL_TO_INT(FifoTablefromCNCLine[0]) DO
			FifoTableFromCNCTemp[p, 0] := FifoTableFromCNCLine[8*p+1];
			FifoTableFromCNCTemp[p, 1] := FifoTableFromCNCLine[8*p+2];
			FifoTableFromCNCTemp[p, 2] := FifoTableFromCNCLine[8*p+3];
			FifoTableFromCNCTemp[p, 3] := FifoTableFromCNCLine[8*p+4];
			FifoTableFromCNCTemp[p, 4] := FifoTableFromCNCLine[8*p+5];
			FifoTableFromCNCTemp[p, 5] := FifoTableFromCNCLine[8*p+6];
			FifoTableFromCNCTemp[p, 6] := FifoTableFromCNCLine[8*p+7];
			FifoTableFromCNCTemp[p, 7] := FifoTableFromCNCLine[8*p+8];
			
		END_FOR
		
		FifoWrite.bExecute := TRUE;
		FifoState := 200;
		FifoHasWritten := FALSE;
		FifoTableCanTakeData := FALSE;
	END_IF
	
200:

	m := m +1;
	FifoWrite.bExecute := FALSE;
	FrameNumber := FrameNumber + 1;
	IF NOT fifostart.bBusy THEN
		//Fifostart.bExecute := TRUE;
		FifoState := 300;
	END_IF
	
300:
	//IF NrOccupiedLines > 0 THEN
		IF NOT fifostart.bBusy then // AND NOT fifostart.bErr THEN
			FifoStart.bExecute := FALSE;
			FifoTableCanTakeData := TRUE;
			Fifostate := 100;
		END_IF
	//END_IF
	
400:
//

500:
	
	//Sätt upp två minnen
	IF FifoTableFromCNC[0,0] <> 0 THEN
		MEMMOVE(ADR(FifoTable2), ADR(FifoTableFromCNC), SIZEOF(FifoTableFromCNC));	
		MEMSET(ADR(FifoTableFromCNC), 0, SIZEOF(FifoTableFromCNC));
	END_IF


END_CASE



CASE FiFoRunState OF

0: 
	IF 	NrOccupiedLines > 0 THEN
		FifoStart.bExecute := TRUE;
	ELSE
			FifoStart.bExecute := FALSE;	
	END_IF

END_CASE


//override
FifoOverride(
	iChannelId:= 2, 
	iOverride:= nOverride, 
	bExecute:= , 
	tTimeout:= T#1S, 
	bBusy=> , 
	bErr=> , 
	iErrId=> );
	
	
fbMethods();


//Integrate
CASE StartInt OF
	0:
	IF StartIntegration THEN
		FOR n:= 1 TO 8 DO
			FIFOChInegrate[n](ChNumber:=(n+9) , PosNumber := n,  bExcute:=TRUE );
		END_FOR
		StartInt := 10;
	END_IF

	10:
	StartIntegration := FALSE;	
	FOR n:= 1 TO 8 DO
		FIFOChInegrate[n](ChNumber:=(n+9) , PosNumber := n,  bExcute:=FALSE );
	END_FOR
	FifoActive := TRUE;
	StartInt := 0;
END_CASE


//Kolla lediga platser
		//läs parametrisering
		FiFoReadDim1(iChannelId:=2 );
		FifoReadDimOK := NOT FiFoReadDim1.bBusy AND NOT FiFoReadDim1.bErr;
		FiFoNoOfAxis := FiFoReadDim1.iNoOfAxes;
		FiFoNoOfEntries := FiFoReadDim1.iNoOfFifoEntries;
		NrOccupiedLines:= MAIN.motor_x_master.Axis.NcToPlc.SafEntries;
		IF FifoActive THEN
			FreeRows := FiFoNoOfEntries - NrOccupiedLines ;
		ELSE
			FreeRows := 0;	
		END_IF
		



//Deintegrate

FifoDeIntegrate(
	iChannelId:= 2, 
	bExecute:= , 
	tTimeout:= , 
	bBusy=> , 
	bErr=> , 
	iErrId=> );
	
	

IF FifoOverride.bExecute THEN
	FifoOverride.bExecute := FALSE;
END_IF

IF FifoDeIntegrate.bExecute THEN
	FifoActive := FALSE;
	FifoDeIntegrate.bExecute := FALSE;
END_IF

FifoWrite(
	iChannelId:= 2, 
	AdrDataArray:= ADR(FifoTableFromCNCTemp), 
	iColDim:= 8, 
	iRowsToWrite:= LREAL_TO_INT(FifoTablefromCNCLine[0]), 
	bExecute:= , 
	tTimeout:= , 
	bBusy=> , 
	bErr=> , 
	iErrId=> );
	
FifoStart(
	iChannelId:= 2, 
	bExecute:= , 
	tTimeout:= , 
	bBusy=> , 
	bErr=> , 
	iErrId=> );

METHOD M_Deintegrate : BOOL
VAR_INPUT
END_VAR
StartFifo := FALSE;
FifoState := 0;
FifoDeIntegrate.bExecute := TRUE;
END_METHOD

METHOD M_Integrate : BOOL
VAR_INPUT
END_VAR


StartIntegration := TRUE;
END_METHOD

END_PROGRAM

// ---- POUs/FIFOIntegrate.TcPOU
FUNCTION_BLOCK FIFOIntegrate
VAR_INPUT
	ChNumber : UINT;
	PosNumber : UINT;
	bExcute: BOOL;
END_VAR
VAR_OUTPUT
	bBusy : BOOL;
	bError : BOOL;
END_VAR
VAR
	FifoIntegrate : FiFoGroupIntegrate;

END_VAR



FifoIntegrate(
	iChannelId:= 2, 
	iAxisId:= ChNumber, 
	iGroupPosition:= PosNumber, 
	bExecute:= bExcute, 
	tTimeout:= , 
	bBusy=> bBusy, 
	bErr=> bError, 
	iErrId=> );

END_FUNCTION_BLOCK

// ---- POUs/FB_methods.TcPOU
FUNCTION_BLOCK FB_methods
VAR_INPUT
END_VAR
VAR_OUTPUT
	StartIntegration : BOOL;
END_VAR
VAR
END_VAR


IF StartIntegration THEN
	FIFOaxis.M_Integrate();
	StartIntegration := FALSE;
END_IF

{attribute 'TcRpcEnable'}
METHOD M_Integrate : BOOL
VAR_INPUT
END_VAR

StartIntegration := TRUE;
END_METHOD

END_FUNCTION_BLOCK

// ---- POUs/IO.TcPOU
PROGRAM IO
VAR
	DI1 AT %I* : BOOL;	// Reset EMC
	DI2 AT %I* : BOOL;	
	DI3 AT %I* : BOOL;
	DI4 AT %I* : BOOL;	
	DI5 AT %I* : BOOL;	
	DI6 AT %I* : BOOL;
	DI7 AT %I* : BOOL;	
	DI8 AT %I* : BOOL;	
	DI9 AT %I* : BOOL;
	DI10 AT %I* : BOOL;
	DI11 AT %I* : BOOL;
	DI12 AT %I* : BOOL;
	DI13 AT %I* : BOOL;
	DI14 AT %I* : BOOL;
	DI15 AT %I* : BOOL;
	DI16 AT %I* : BOOL;
	DI17 AT %I* : BOOL;
	DI18 AT %I* : BOOL;
	DI19 AT %I* : BOOL;
	DI20 AT %I* : BOOL;
	DI21 AT %I* : BOOL;
	DI22 AT %I* : BOOL;
	DI23 AT %I* : BOOL;
	DI24 AT %I* : BOOL;
	DI25 AT %I* : BOOL;
	DI26 AT %I* : BOOL;
	DI27 AT %I* : BOOL;
	DI28 AT %I* : BOOL;

	
	DOs : ARRAY[1..64] OF DigitalOut;
	
	ArrayData1 : ARRAY[0..50] OF ST_streamOutputs;
	ArrayData2 : ARRAY[0..50] OF ST_streamOutputs;
	
	AI1 AT %I* : INT;
	AI2 AT %I* : INT;
	AI3 AT %I* : INT;
	
	AO1 AT %Q* : INT;
	AO2 AT %Q* : INT;
	AO3 AT %Q* : INT;

	newStreamData: BOOL;
	cycleCounter2ms: UINT;
	startStream: BOOL;
	i: INT;
	
	counterValue AT %I* : UINT;
	EMCOK  AT %I*:BOOL;
	EMCDelayedOK  AT %I*:BOOL;
	Run  AT %Q* :BOOL:=TRUE;
	AckSaftey  AT %Q*:BOOL;
	ResetSaftey AT%Q*:BOOL;
	state: INT;
	bIsResetting: BOOL;
	
	bBlueLight AT  %Q*:BOOL;

END_VAR



FOR i:= 1 TO 64 DO
	DOs[i]();
END_FOR




IF DI1 OR bIsResetting THEN
	CASE state OF 
		
	 0:		Run:=FALSE;
			AckSaftey:=FALSE;
	 		ResetSaftey:=FALSE;
			bIsResetting:=TRUE;
			state:=10;
	 
	 10:	AckSaftey:=TRUE;
	 		state:=20;
			
	20: AckSaftey:=FALSE; // Finnished
		
		state:=25;
	25:
		Run:=TRUE;
		state:=30;
	30: ResetSaftey:=TRUE;
		state:=40;
	40: // Finnished
	
	dI1:= bIsResetting:=FALSE;
	ResetSaftey:=FALSE;
	 state:=0;
	 
	
	END_CASE

END_IF

bBlueLight := NOT EMCOK;

END_PROGRAM

// ---- POUs/DigitalOut.TcPOU
FUNCTION_BLOCK DigitalOut
VAR_INPUT
END_VAR
VAR_OUTPUT
END_VAR
VAR
	DO_io  AT %Q*: BOOL;
	timerOn : TON;
	timerOff : TON;
	onActive : BOOL;
	offActive : BOOL;
	Do_in: BOOL;
	ActualCycle : UDINT;
	fbGetCurrTask : GETCURTASKINDEX;
	NextOn: UDINT;
	NextOff :UDINT;
	fifo : FB_Fifo;
	NextOnOff : ST_streamOutputs;
	init: BOOL;
END_VAR


IF init THEN
	init := FALSE;
	fifo.M_init();
	NextOnoff.cycleNo := 0;
END_IF



ActualCycle := TwinCAT_SystemInfoVarList._TaskInfo[1].CycleCount;
fifo();



IF fifo.bDataInBuffer AND NextOnOff.cycleNo = 0 THEN
	NextOnOff := fifo.M_RemoveEntry();
END_IF


IF ActualCycle = NextOnOff.cycleNo THEN
	NextOnOff.cycleNo := 0;
	DO_io := nextonoff.on;
END_IF

{attribute 'TcRpcEnable'}
METHOD M_OffWithDelay : BOOL
VAR_INPUT
	cycleNo : INT;
END_VAR

VAR

END_VAR



NextOff := ActualCycle + cycleNo + FIFOaxis.NrOccupiedLines;


fifo.M_AddEntry(NextOff, FALSE);
END_METHOD

{attribute 'TcRpcEnable'}
METHOD M_OnWithDelay : BOOL
VAR_INPUT
	cycleNo : INT;
END_VAR

VAR

END_VAR


NextOn := ActualCycle + cycleNo + FIFOaxis.NrOccupiedLines;

fifo.M_AddEntry(NextOn, TRUE);
END_METHOD

END_FUNCTION_BLOCK

// ---- POUs/FB_Fifo.TcPOU
FUNCTION_BLOCK FB_Fifo
VAR CONSTANT
	NoOfEntries: INT := 100;
END_VAR
VAR_INPUT
END_VAR
VAR_OUTPUT
	bDataInBuffer: BOOL;
	bBufferFull: BOOL;
	MaxBuffer : INT;
END_VAR
VAR
	Buffer : ARRAY[0..NoOfEntries] OF ST_streamOutputs;
	init: BOOL := true;
	index: INT;
END_VAR


IF init THEN
	index := 0;
	MaxBuffer := 0;
	init := FALSE;
END_IF

bDataInBuffer := index > 0;
bBufferFull := index >= NoOfEntries;


IF index > MaxBuffer THEN
	Maxbuffer := index;
END_IF

METHOD M_AddEntry : BOOL
VAR_INPUT
	cycleNo : UDINT;
	on : BOOL;

END_VAR
VAR_OUTPUT
	bError: BOOL;
END_VAR
VAR
		stEntry : ST_streamOutputs;
END_VAR

IF (index < NoOfEntries) THEN
	stEntry.cycleNo := cycleNo;
	stEntry.on := on;
	
	Buffer[index] := stEntry;
	index := index + 1;
	M_AddEntry :=TRUE;
	bError := FALSE;
ELSE
	bError := TRUE;	
END_IF
END_METHOD

METHOD M_init : BOOL
VAR_INPUT
END_VAR
init := true;
END_METHOD

METHOD M_RemoveEntry : ST_streamOutputs
VAR_INPUT
END_VAR

VAR
	n: INT;
END_VAR


IF (index > 0) THEN
	M_RemoveEntry := Buffer[0];

	MEMCPY(destAddr:= ADR(Buffer[0]), srcAddr:=ADR(Buffer[1]), n:=(SIZEOF(Buffer)-SIZEOF(Buffer[1])));
	MEMSET(ADR(Buffer[index]), 0, SIZEOF(Buffer[index]));
	index := index -1;

END_IF
END_METHOD

END_FUNCTION_BLOCK
